(* IEC 61131-3 sources: UserLog/, 5 files *)

(* ---- Types.typ ---- *)
TYPE
	UserLogErrorEnum :
		(
		USERLOG_ERROR_NONE := 0,
		USERLOG_ERROR_INVALID_SEVERITY := 101, (*The severity is not an option when generating the EventID (<= 3)*)
		USERLOG_ERROR_TASK_NAME, (*The task name function from sys_lib has returned an error*)
		USERLOG_ERROR_LOGBOOK_IDENT, (*The function block to retrieve the user logbook ident address has returned an error*)
		USERLOG_ERROR_WRITE, (*The function block to write an entry to the user logbook has returned an error*)
		USERLOG_ERROR_BUFFER_FULL (*The log buffer is full and no further events can be written until the buffer is emptied*)
		);
	UserLogSeverityEnum :
		( (*Levels of severity, see AS Help 32-bit event ID*)
		USER_LOG_SEVERITY_SUCCESS := 0, (*The logbook entry marks success operation completion*)
		USER_LOG_SEVERITY_INFORMATION := 1, (*An informative entry useful to the user*)
		USER_LOG_SEVERITY_WARNING := 2, (*An issue has occured during operation but is not critical*)
		USER_LOG_SEVERITY_ERROR := 3 (*An error has occured during operation*)
		);
	UserLogCyclicStateEnum :
		(
		USER_LOG_STATE_INIT,
		USER_LOG_STATE_IDENT,
		USER_LOG_STATE_IDLE,
		USER_LOG_STATE_WRITE,
		USER_LOG_STATE_ERROR := 255
		);
	UserLogBufferInfoType : 	STRUCT
		WriteIndex : USINT;
		ReadIndex : USINT;
		Full : BOOL;
		State : UserLogCyclicStateEnum;
		UserLogbookIdent : ArEventLogIdentType;
		NumEntriesInBuffer : USINT;
		NumEntriesLogged : USINT;
		NumEntriesLost : USINT;
	END_STRUCT;
END_TYPE

(* ---- UserLog.typ ---- *)
(*******************************************************************************
 * File: UserLog.typ
 * Author: Tyler Matijevich
 * Created: 2020-10-29
*******************************************************************************)

TYPE
	UserLogSeverityEnum :
		( (*Levels of severity. See 32-bit event ID in help*)
		USERLOG_SEVERITY_DEBUG := -1, (*Information: Developer information*)
		USERLOG_SEVERITY_SUCCESS, (*Success: Completion*)
		USERLOG_SEVERITY_INFORMATION, (*Information: User information*)
		USERLOG_SEVERITY_WARNING, (*Warning: The application may continue*)
		USERLOG_SEVERITY_ERROR, (*Error: The application in recoverable*)
		USERLOG_SEVERITY_CRITICAL (*Error: The application in unrecoverable*)
		);
	UserLogFormatType : 	STRUCT  (*Argument structure for runtime format data*)
		b : ARRAY[0..USERLOG_FORMAT_INDEX]OF BOOL; (*Place boolean (TRUE or FALSE)*)
		f : ARRAY[0..USERLOG_FORMAT_INDEX]OF LREAL; (*Place double*)
		i : ARRAY[0..USERLOG_FORMAT_INDEX]OF DINT; (*Place integer (32-bit signed)*)
		s : ARRAY[0..USERLOG_FORMAT_INDEX]OF STRING[USERLOG_FORMAT_LENGTH]; (*Place string*)
	END_STRUCT;
END_TYPE

(* ---- UserLog.fun ---- *)
FUNCTION UserLogBasic : UDINT (*Write to the User logbook synchronously*)
	VAR_INPUT
		Severity : DINT; (*Use UserLogSeverityEnum or arEVENTLOG_SEVERITY constants*)
		Code : UINT; (*0..65535*)
		Message : STRING[0]; (*Event description*)
	END_VAR
END_FUNCTION

FUNCTION UserLogAdvanced : UDINT (*Write to the User logbook with runtime data*)
	VAR_INPUT
		Severity : DINT; (*Use UserLogSeverityEnum or arEVENTLOG_SEVERITY constants*)
		Code : UINT; (*0..65535*)
		Message : STRING[0]; (*Event description with optional format specifiers*)
		Values : UserLogFormatType; (*Format values to replace specifiers (%b, %f, %i, %s)*)
	END_VAR
END_FUNCTION

FUNCTION UserLogCustom : UDINT (*Write to any user logbook synchronously*)
	VAR_INPUT
		Logbook : STRING[0]; (*Name of logbook*)
		Severity : DINT; (*Use UserLogSeverityEnum or arEVENTLOG_SEVERITY constants*)
		Facility : UINT; (*0..4095*)
		Code : UINT; (*0..65535*)
		Origin : ArEventLogRecordIDType; (*(Optional) Origin record ID*)
		Object : STRING[0]; (*(Optional) Object name*)
		Message : STRING[0]; (*Event description with optional format specifiers*)
		Values : UserLogFormatType; (*Format values to replace specifiers (%b, %f, %i, %s)*)
	END_VAR
END_FUNCTION

FUNCTION UserLogEventText : UDINT (*Write to any user logbook through binary-encoded data and event texts*)
	VAR_INPUT
		Logbook : STRING[0]; (*Name of logbook*)
		Event : DINT; (*Event ID (match Text ID)*)
		Origin : ArEventLogRecordIDType; (*(Optional) Origin record ID*)
		Object : STRING[0]; (*(Optional) Object name*)
		Message : STRING[0]; (*Event description with optional format specifiers*)
		Values : UserLogFormatType; (*Format values to replace specifiers (%b, %f, %i, %s)*)
	END_VAR
END_FUNCTION

FUNCTION UserLogCreate : DINT (*Create a custom logbook in an Init subroutine*)
	VAR_INPUT
		Name : STRING[0]; (*Name of logbook limited to 10 characters*)
		Size : UDINT; (*Size of logbook in bytes (minimum 4096)*)
	END_VAR
END_FUNCTION

FUNCTION UserLogSetSeverityLevel : DINT (*Suppress messages below the input level and return previous level*)
	VAR_INPUT
		Level : DINT; (*Severity level threshold*)
	END_VAR
END_FUNCTION

FUNCTION UserLogGetSeverity : USINT (*Get ArEventLog severity from an event ID*)
	VAR_INPUT
		Event : DINT; (*Event ID*)
	END_VAR
END_FUNCTION

FUNCTION UserLogGetFacility : UINT (*Get ArEventLog facility from an event ID*)
	VAR_INPUT
		Event : DINT; (*Event ID*)
	END_VAR
END_FUNCTION

FUNCTION UserLogGetCode : UINT (*Get ArEventLog code from an event ID*)
	VAR_INPUT
		Event : DINT; (*Event ID*)
	END_VAR
END_FUNCTION

(* ---- Constants.var ---- *)
VAR CONSTANT
	USER_LOG_BUFFER_SIZE : USINT := 250; (*Number of buffered entries for writing to the user logbook*)
	USER_LOG_MESSAGE_LENGTH : USINT := 125; (*String length of the formatted messages written to the logger*)
	USER_LOG_MAX_INDEX_BUFFER : USINT := USER_LOG_BUFFER_SIZE -1; (*Size of buffer minus one for IEC variable declaration*)
END_VAR

(* ---- UserLog.var ---- *)
VAR CONSTANT
	USERLOG_MESSAGE_LENGTH : UDINT := 120; (*Maximum length of all messages written to user logbooks*)
	USERLOG_FACILITY : UINT := 10; (*Facility number used for UserLogBasic and UserLogAdvanced functions*)
	USERLOG_ERROR_IDENT : DINT := -515234032; (*An error occurred when calling ArEventLogGetIdent. See User logbook for details*)
	USERLOG_ERROR_WRITE : DINT := -515234022; (*An error occurred when calling ArEventLogWrite. See User logbook for details*)
	USERLOG_ERROR_CREATE : DINT := -515234012; (*An error occurred when calling ArEventLogCreate. See User logbook for details*)
	USERLOG_FORMAT_INDEX : USINT := 5; (*Maximum index of each runtime data type*)
	USERLOG_FORMAT_LENGTH : USINT := 80; (*Length of string runtime data*)
	USERLOG_EXAMPLE_TEXT_ID : DINT := 1632259616; (*Example Text ID (Event ID) for UserLogEventText function*)
END_VAR
